PROGRAM MAIN
VAR
END_VAR

END_PROGRAM

(* stored: Version 1.1.0.1
   POU MAIN: Id {8ad25079-75c3-46d0-aa3a-e257b640d76a} *)
